// TwinCAT 3 PLC project EventLib
// ProgramVersion: 3.1.4023.0
// libraries:
//   Tc2_Standard, * (Beckhoff Automation GmbH)
//   Tc2_System, * (Beckhoff Automation GmbH)
//   Tc3_EventLogger, * (Beckhoff Automation GmbH)
//   Tc3_Module, * (Beckhoff Automation GmbH)
// project tree:
//   EventLoggerClass/ ITcMessage_Ext.TcIO, TcMessage_Ext.TcPOU
//   / PlcTask.TcTTO
//   POUs/ MAIN.TcPOU

CONFIGURATION EventLib
    RESOURCE PLC ON TwinCAT3
        TASK PlcTask(INTERVAL := T#10ms, PRIORITY := 20);
        PROGRAM MAIN WITH PlcTask : MAIN;
    END_RESOURCE
END_CONFIGURATION

// ---- EventLoggerClass/ITcMessage_Ext.TcIO
INTERFACE ITcMessage_Ext

METHOD Send : BOOL
VAR_INPUT
	eventType : Tc3_EventLogger.TcEventEntry;
	args : STRING(255);
END_VAR
END_METHOD

END_INTERFACE

// ---- POUs/MAIN.TcPOU
PROGRAM MAIN
VAR
END_VAR

END_PROGRAM

// ---- EventLoggerClass/TcMessage_Ext.TcPOU
FUNCTION_BLOCK TcMessage_Ext IMPLEMENTS ITcMessage_Ext
VAR_INPUT
END_VAR
VAR_OUTPUT
END_VAR
VAR
    fbMsg : FB_TcMessage; 
	fbTest : Tc3_EventLogger.FB_TcEvent;
	fbInfo : Tc3_EventLogger.FB_TcSourceInfo;
	_loggerLevel : TcEventSeverity := TcEventSeverity.Info;
END_VAR

PROPERTY PUBLIC LoggerLevel : TcEventSeverity
GET
LoggerLevel := _loggerLevel;
END_GET
SET
_loggerLevel := LoggerLevel;
END_SET
END_PROPERTY

METHOD PUBLIC Send : BOOL
VAR_INPUT
	eventType : Tc3_EventLogger.TcEventEntry;
	args : STRING(255);
END_VAR
IF eventType.eSeverity >= LoggerLevel THEN
	THIS^.fbMsg.CreateEx(eventType, 0);
	THIS^.fbMsg.ipArguments.AddString(args);
	THIS^.fbMsg.Send(0);
	THIS^.fbMsg.Release();
END_IF
END_METHOD

END_FUNCTION_BLOCK
